// TIA Portal V19 export
TYPE "LEXCHANGETRAY_typePlasticEm5_recieve_interface"
// stored: Access Published
   STRUCT
      roller { S7_SetPoint := 'True'} : "LEXCHANGETRAY_typePlasticEm5_toRollerRecieve";
      handlingXyz { S7_SetPoint := 'True'} : "LEXCHANGETRAY_typePlasticEm5_toHandlingXyzRecieve";
   END_STRUCT;
END_TYPE
